(* CoDeSys 2.3.9.28 project: Aula15_ex.pro *)
(* Libraries: Standard.lib 27.1.09 11:27:38, Util.lib 27.1.09 11:27:38, IecSfc.lib 24.11.08 08:07:15, SysLibTime.lib 27.1.09 11:27:38, SysTaskInfo.lib 24.11.08 08:07:15, SYSLIBCALLBACK.LIB 27.1.09 11:27:38 *)

(* PLC configuration (modules and I/O channels)
CPX-CEC [Root] node -1, in %IB0 out %QB0 {StringParam = 2773,0,0,0,0; ByteParam = 0; ByteParam = 31; ByteParam = 0; ByteParam = 0; ByteParam = 0; ByteParam = 0; ByteParam = 0; ByteParam = 0; ByteParam = 2; ByteParam = 0; ByteParam = 0; ByteParam = 0; ByteParam = 32; ByteParam = 0; ByteParam = 0; ByteParam = 5; ByteParam = 0; ByteParam = 0; ByteParam = 0; ByteParam = 0; ByteParam = 0; ByteParam = 0; ByteParam = 0; ByteParam = 0; ByteParam = 14; ByteParam = 240; ByteParam = 192; ByteParam = 168; ByteParam = 2; ByteParam = 10; ByteParam = 255; ByteParam = 255; ByteParam = 0; ByteParam = 0; ByteParam = 192; ByteParam = 168; ByteParam = 1; ByteParam = 1; ByteParam = 192; ByteParam = 168; ByteParam = 2; ByteParam = 10; ByteParam = 255; ByteParam = 255; ByteParam = 0; ByteParam = 0; ByteParam = 192; ByteParam = 168; ByteParam = 1; ByteParam = 1}
  Hexswitch AT %IB0 [HexSwitch] rotary switch 0 = STOP, 1-15 = RUN
  IOModules [CPX_MASTER] node 0, in %IB4 out %QB0
*)

(* Global variable list: Global_Variables *)
VAR_GLOBAL

	START: BOOL;
	STOP: BOOL;
	S1: BOOL;
	S2: BOOL;
	S3: BOOL;

	M1: BOOL;
	C1: BOOL;
	LP: BOOL;
	V1: BOOL;

	MEM2: BOOL;
	MEM3: BOOL;

	T3 : TON;

	PISCA_PISCA : PISCA_LED;

END_VAR

(* POU PLC_PRG, ST *)
PROGRAM PLC_PRG
VAR

END_VAR
T3(IN:= S2 AND MEM2, PT:=T#5S);
PISCA_PISCA(LIGA := LP, DESLIGA := STOP OR (S3 AND MEM3));



IF START THEN
	M1 := TRUE;
	C1 := TRUE;
	LP := TRUE;
END_IF


IF S1 THEN
	C1 := FALSE;
	MEM2 := TRUE;
END_IF


IF S2 AND MEM2 THEN
	M1 := FALSE;
	V1 := TRUE;
END_IF


IF T3.Q THEN
	V1 := FALSE;
	M1 := TRUE;
	MEM2 := FALSE;
	MEM3 := TRUE;
END_IF


IF S3 AND MEM3 THEN
	M1 := FALSE;
	C1 := FALSE;
	V1 := FALSE;
	MEM3 := FALSE;
	LP := FALSE;
END_IF


IF STOP THEN
	M1 := FALSE;
	C1 := FALSE;
	V1 := FALSE;
	MEM2 := FALSE;
	MEM3 := FALSE;
	LP := FALSE;
END_IF
END_PROGRAM

(* POU PISCA_LED, ST *)
FUNCTION_BLOCK PISCA_LED
VAR_INPUT
	LIGA : BOOL;
	DESLIGA : BOOL;
END_VAR
VAR_OUTPUT
	SAIDA : BOOL;
END_VAR
VAR
	T1 : TON;
	T2 : TON;
	MEM : BOOL;
END_VAR
T1(IN:=LP, PT:=T#1S);
T2(IN:= NOT LP, PT:=T#1S);

IF LIGA AND T1.Q AND NOT MEM THEN
	LP := FALSE;
END_IF


IF NOT LIGA AND  T2.Q AND NOT MEM THEN
	LP := TRUE;
END_IF


IF DESLIGA THEN
	MEM := TRUE;
END_IF

IF LIGA THEN
	MEM := FALSE;
END_IF
END_FUNCTION_BLOCK

(* Visualisation screen
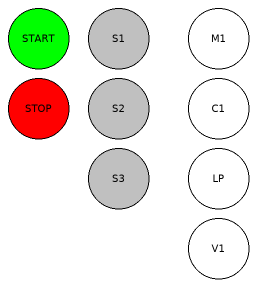
ellipse at (130,50)-(191,111): text "S1"; alarm colour if S1; taps S1
ellipse at (130,120)-(191,181): text "S2"; alarm colour if S2; toggles S2
ellipse at (130,190)-(191,251): text "S3"; alarm colour if S3; taps S3
ellipse at (50,50)-(111,111): text "START"; alarm colour if START; taps START
ellipse at (50,120)-(111,181): text "STOP"; alarm colour if STOP; taps STOP
ellipse at (230,120)-(291,181): text "C1"; alarm colour if C1
ellipse at (230,190)-(291,251): text "LP"; alarm colour if LP
ellipse at (230,260)-(291,321): text "V1"; alarm colour if V1
ellipse at (230,50)-(291,111): text "M1"; alarm colour if M1
*)
